INTERFACE IRunner

METHOD registerTestSuite
VAR_INPUT
    testSuite: ITestSuite;
END_VAR
END_METHOD

END_INTERFACE

(* stored: Version 1.1.0.1, ProductVersion 3.1.4022.12
   Itf IRunner: Id {7785b053-0144-45ae-90de-76fa438cd345}
   Method registerTestSuite: Id {1614c136-9cec-47d8-8bb5-5e9b535bff2a} *)
